// TIA Portal V17 export
// export: Created 2025-03-12T15:37:54.9879156Z, ExportSetting WithDefaults, DisplayName Totally Integrated Automation Portal, DisplayVersion V17 Update 8, DisplayName TIA Portal Openness, DisplayVersion V17 Update 8, DisplayName TIA Portal Version Control Interface, DisplayVersion V17, DisplayName SINAMICS Startdrive Advanced, DisplayVersion V17 SP2, DisplayName SINAMICS Startdrive G110M, G120, G120C, G120D, G120P, G115D, DisplayVersion V17 SP2, DisplayName SINAMICS Startdrive G130, G150, S120, S150, SINAMICS MV, S210, DisplayVersion V17 SP2, DisplayName STEP 7 Professional, DisplayVersion V17 Update 8, DisplayName SINUMERIK ONE STEP 7 Toolbox, DisplayVersion V17 Update 12, DisplayName SINUMERIK 840D sl STEP 7 Toolbox, DisplayVersion V17 Update 12, DisplayName STEP 7 Safety, DisplayVersion V17 Update 6, DisplayName WinCC Advanced, DisplayVersion V17 Update 8
TYPE "SAFETY_GROUP"
// stored: IsFailsafeCompliant true
   STRUCT
      STO_Deactivate : Bool;   // SAFE TORQUE OFF DEACTIVATE
      SS1_Deactivate : Bool;   // SAFE STOP 1 DEACTIVATE
      SS2_Deactivate : Bool;   // SAFE STOP 2 DEACTIVATE
      SS2E_Deactivate : Bool;   // SAFE STOP 2 EXTENDED DEACTIVATE
      SOS_Deactivate : Bool;   // SAFE OPERATING STOP DEACTIVATE
      SLS_Deactivate : Bool;   // SAFE LIMITED SPEED DEACTIVATE
      SLS_BIT0 : Bool;   // SAFE LIMITED SPEED BIT 0
      SLS_BIT1 : Bool;   // SAFE LIMITED SPEED BIT 1
   END_STRUCT;
END_TYPE
